TYPE EventMessage :
STRUCT
  id: INT;
  path: STRING(255);
  message: STRING(255);
  level: EventLevel;
  cleared: BOOL;
END_STRUCT
END_TYPE

(* stored: Version 1.1.0.1, ProductVersion 3.1.4024.9
   DUT EventMessage: Id {eab319f3-c899-4cf2-8754-0b17b4d9d8d7} *)
